ABB RAPID module: 00094CE0

MODULE Module1
    PERS tooldata Sopapa:=[TRUE,[[0,-5,103],[1,0,0,0]],[.500,[0,0,40],[1,0,0,0],0,0,0]];
    CONST robtarget Target_10:=[[595.492267836,-5,628],[0.5,0,0.866025404,0],[0,0,0,0],[9E+09,9E+09,9E+09,9E+09,9E+09,9E+09]];
    CONST robtarget Target_20:=[[595.492192643,34.78927249,628.000011052],[0.500000018,0.000000003,0.866025394,0.000000005],[0,-1,0,0],[9E+09,9E+09,9E+09,9E+09,9E+09,9E+09]];
!***********************************************************
    !
    ! Module:  Module1
    !
    ! Description:
    !   <Insert description here>
    !
    ! Author: CARTELLI
    !
    ! Version: 1.0
    !
    !***********************************************************


    !***********************************************************
    !
    ! Procedure main
    !
    !   This is the entry point of your program
    !
    !***********************************************************
    PROC main()
        !Add your code here
        Path_10;
    ENDPROC
    PROC Path_10()
        MoveL Target_10,v1000,z100,Sopapa\WObj:=wobj0;
        MoveL Target_20,v1000,z100,Sopapa\WObj:=wobj0;
    ENDPROC
ENDMODULE
